// TIA Portal project "Hardware" (V14)

(* hardware
DEVICE "ET 200S-Station_1"  ET 200S station
   slot 0: "Baugruppenträger_0"  Rail
   slot 2: "PLC_1"  IM151-8 CPU  6ES7 151-8AB00-0AB0  V2.7
      slot 1: "PROFINET-Schnittstelle_1"  PN-IO
         slot 1: "Port_1"  Port
         slot 2: "Port_2"  Port
         slot 3: "Port_3"  Port
   slot 4: "PM-E 24VDC_1"  PM-E 24VDC  6ES7 138-4CA01-0AA0
   slot 5: "4AI x I 2WIRE ST_1"  4AI x I 2WIRE ST  6ES7 134-4GD00-0AB0
   slot 6: "2AO x U ST_1"  2AO x U ST  6ES7 135-4FB01-0AB0
   slot 7: "8DI x 24VDC_1"  8DI x 24VDC  6ES7 131-4BF00-0AA0
   slot 8: "8DI x 24VDC_2"  8DI x 24VDC  6ES7 131-4BF00-0AA0
   slot 9: "8DI x 24VDC_3"  8DI x 24VDC  6ES7 131-4BF00-0AA0
   slot 10: "8DI x 24VDC_4"  8DI x 24VDC  6ES7 131-4BF00-0AA0
   slot 11: "8DO x 24VDC / 0.5A_1"  8DO x 24VDC / 0.5A  6ES7 132-4BF00-0AA0
   slot 12: "8DO x 24VDC / 0.5A_2"  8DO x 24VDC / 0.5A  6ES7 132-4BF00-0AA0
   slot 13: "8DO x 24VDC / 0.5A_3"  8DO x 24VDC / 0.5A  6ES7 132-4BF00-0AA0
   slot 14: "8DO x 24VDC / 0.5A_4"  8DO x 24VDC / 0.5A  6ES7 132-4BF00-0AA0
DEVICE "HMI_1"  TP 177B 6'' PN/DP
   slot 0: "TP 177B 6'' PN/DP"  TP 177B 6'' PN/DP  6AV6 642-0BA01-1AX1  11.0.2.0
   slot 1: "HMI_RT_1"  TP 177B 6'' PN/DP  6AV6 642-0BA01-1AX1  11.0.2.0
   slot 5: "HMI_1.IE_CP_1"  PROFINET Interface  11.0.0.0
      slot 1: "PROFINET Schnittstelle_1"  PROFINET Interface
         slot 1: "Port_1"  Port
   slot 7: "HMI_1.MPI/DP_CP_1"  MPI/DP Interface  11.0.0.0
DEVICE "S7-1200-Station_1"  S7-1200 Station
   slot 0: "Baugruppenträger_0"  S7-1200 Rack  Rack  V1.0
   slot 1: "PLC_2"  CPU 1214FC DC/DC/DC  6ES7 214-1AF40-0XB0  V4.2
   slot 2: "F-DI 8/16x24VDC_1"  SM 1226 F-DI8/16 x 24VDC  6ES7 226-6BA32-0XB0  V2.0
   slot 3: "AI 1xRTD_1"  AI1 x RTD signal board  6ES7 231-5PA30-0XB0  V2.0
   slot 3: "F-DQ 4x24VDC_1"  SM 1226 F-DQ4 x 24VDC  6ES7 226-6DA32-0XB0  V2.0
   slot 4: "AI 4x13BIT/AQ 2x14BIT_1"  6ES7 234-4HE32-0XB0  V2.0
*)

// ===== PLC "PLC_1"  IM151-8 CPU =====

VAR_GLOBAL   // PLC tag table "Standard-Variablentabelle"
   "Blinken" AT %A7.0 : Bool;
   "Sekundentakt" AT %M100.5 : Bool;
   "A_rot" AT %A9.6 : Bool;
   "A_gelb" AT %A9.7 : Bool;
   "A_gruen" AT %A10.0 : Bool;
   "F_rot" AT %A10.6 : Bool;
   "F_gruen" AT %A10.7 : Bool;
   "Tag_1" AT %M0.0 : Bool;
   "Zweisekundentakt" AT %M100.7 : Bool;
   "Tag_2" AT %M3.0 : Bool;
   "Tag_3" AT %MD12 : DWord;
   "Tag_4" AT %MD16 : DWord;
   "Tag_5" AT %MW20 : Int;
   "Tag_6" AT %MW21 : Int;
   "Tag_7" AT %MW30 : Int;
   "Tag_8" AT %M22.7 : Bool;
   "Tag_9" AT %M2.0 : Bool;
   "Tag_10" AT %EW272 : Int;
END_VAR

DATA_BLOCK "Tagbetrieb_fb_DB"   // DB2
{ S7_Optimized_Access := 'FALSE' }
VERSION : 0.1
// stored: InstanceOfName Tagbetrieb_fb
"Tagbetrieb_fb"
BEGIN
END_DATA_BLOCK

DATA_BLOCK "DB3_Farben"   // DB3
{ S7_Optimized_Access := 'FALSE' }
VERSION : 0.1
   VAR
      rot : Int;
      gruen : Int;
      blau : Int;
   END_VAR
BEGIN
END_DATA_BLOCK

DATA_BLOCK "Farben"   // DB4
{ S7_Optimized_Access := 'FALSE' }
VERSION : 0.1
   VAR
      Farben : Array[0..2, 0..9] of Real;
      Rot : Real;
      Blau : Real;
      Gelb : Real;
      index : Int;
      schreiben : Bool;
   END_VAR
BEGIN
END_DATA_BLOCK

DATA_BLOCK "Zu_1200"   // DB100
{ S7_Optimized_Access := 'FALSE' }
VERSION : 0.1
   VAR
      Gewicht_rot : Real;
      Gewicht_Gruen : Real;
      Gewicht_Blau : Real;
   END_VAR
BEGIN
END_DATA_BLOCK

DATA_BLOCK "Von_1200"   // DB101
{ S7_Optimized_Access := 'FALSE' }
VERSION : 0.1
   VAR
      Temperatur : Int;
   END_VAR
BEGIN
END_DATA_BLOCK

DATA_BLOCK "Variable"   // DB200
{ S7_Optimized_Access := 'FALSE' }
VERSION : 0.1
   VAR
      Abstand : Real;
      Gewicht_real : Real;
      Volumen : Real;
      Tag : Bool;
      Zeit : Int;
      Tag_H : Int;
      Tag_M : Int;
      Start_tag : Int;
      Nacht_H : Int;
      Nacht_M : Int;
      Start_Nacht : Int;
   END_VAR
BEGIN
END_DATA_BLOCK

FUNCTION_BLOCK "Tagbetrieb_fb"   // FB1, FBD
{ S7_Optimized_Access := 'FALSE' }
VERSION : 0.1
   VAR_INPUT
      Sekundentakt : Bool;
   END_VAR
   VAR_OUTPUT
      Auto_rot : Bool;
      Auto_gelb : Bool;
      Auto_gruen : Bool;
      FG_rot : Bool;
      FG_gruen : Bool;
   END_VAR
   VAR
      S5 : Bool;
   END_VAR
   VAR_TEMP
      S1 : Bool;
      S2 : Bool;
      S3 : Bool;
      S4 : Bool;
      Zaehler : Int;
   END_VAR
BEGIN

REGION Network 1
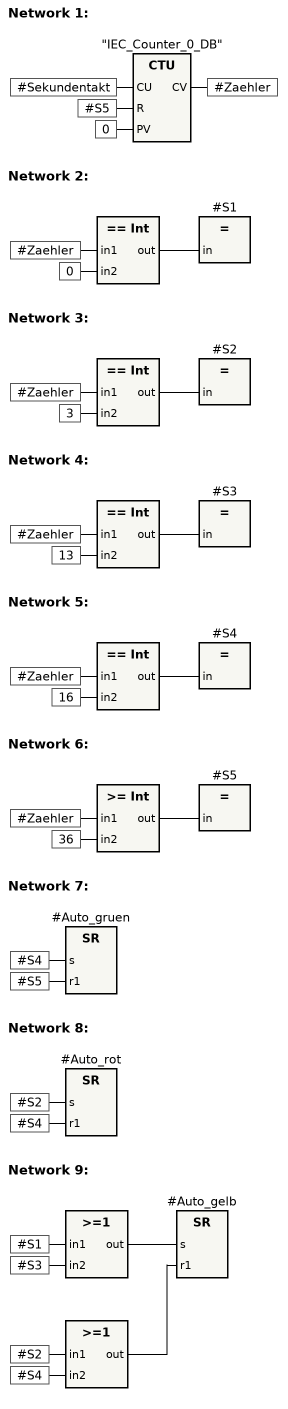
   "IEC_Counter_0_DB".CTU(CU := #Sekundentakt, R := #S5, PV := 0, CV => #Zaehler);
END_REGION

REGION Network 2
   #S1 := #Zaehler = 0;
END_REGION

REGION Network 3
   #S2 := #Zaehler = 3;
END_REGION

REGION Network 4
   #S3 := #Zaehler = 13;
END_REGION

REGION Network 5
   #S4 := #Zaehler = 16;
END_REGION

REGION Network 6
   #S5 := #Zaehler >= 36;
END_REGION

REGION Network 7
   IF #S4 THEN
       #Auto_gruen := TRUE;   // SR flip-flop
   END_IF;
   IF #S5 THEN #Auto_gruen := FALSE; END_IF;
END_REGION

REGION Network 8
   IF #S2 THEN
       #Auto_rot := TRUE;   // SR flip-flop
   END_IF;
   IF #S4 THEN #Auto_rot := FALSE; END_IF;
END_REGION

REGION Network 9
   IF #S1 OR #S3 THEN
       #Auto_gelb := TRUE;   // SR flip-flop
   END_IF;
   IF #S2 OR #S4 THEN #Auto_gelb := FALSE; END_IF;
END_REGION

REGION Network 10
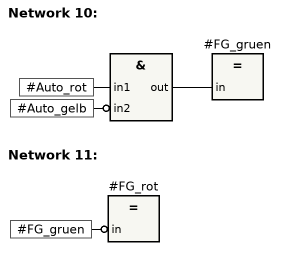
   #FG_gruen := #Auto_rot AND NOT #Auto_gelb;
END_REGION

REGION Network 11
   #FG_rot := NOT #FG_gruen;
END_REGION
END_FUNCTION_BLOCK

FUNCTION "Tagbetrieb" : Void   // FC1, FBD
{ S7_Optimized_Access := 'FALSE' }
VERSION : 0.1
   VAR_INPUT
      Sekundentakt : Bool;
   END_VAR
   VAR_OUTPUT
      Auto_rot : Bool;
      Auto_gelb : Bool;
      Auto_gruen : Bool;
      FG_rot : Bool;
      FG_gruen : Bool;
   END_VAR
   VAR_TEMP
      S1 : Bool;
      S2 : Bool;
      S3 : Bool;
      S4 : Bool;
      S5 : Bool;
      Zaehler : Int;
   END_VAR
BEGIN

REGION Network 1
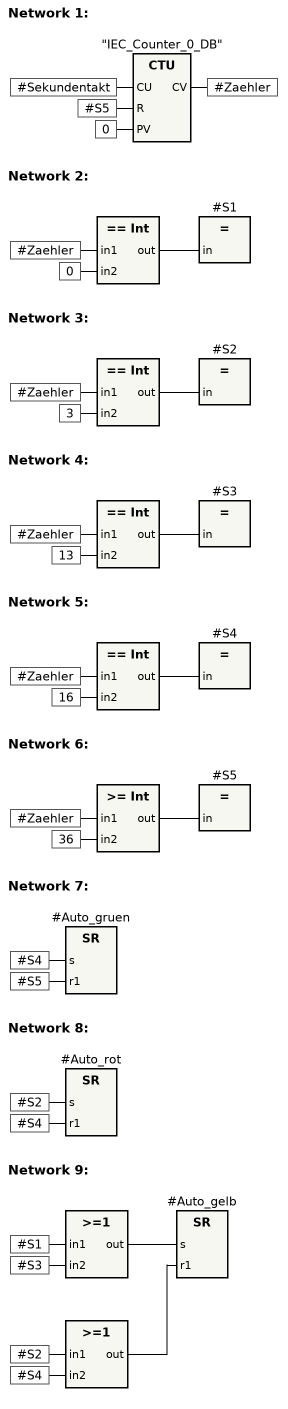
   "IEC_Counter_0_DB".CTU(CU := #Sekundentakt, R := #S5, PV := 0, CV => #Zaehler);
END_REGION

REGION Network 2
   #S1 := #Zaehler = 0;
END_REGION

REGION Network 3
   #S2 := #Zaehler = 3;
END_REGION

REGION Network 4
   #S3 := #Zaehler = 13;
END_REGION

REGION Network 5
   #S4 := #Zaehler = 16;
END_REGION

REGION Network 6
   #S5 := #Zaehler >= 36;
END_REGION

REGION Network 7
   IF #S4 THEN
       #Auto_gruen := TRUE;   // SR flip-flop
   END_IF;
   IF #S5 THEN #Auto_gruen := FALSE; END_IF;
END_REGION

REGION Network 8
   IF #S2 THEN
       #Auto_rot := TRUE;   // SR flip-flop
   END_IF;
   IF #S4 THEN #Auto_rot := FALSE; END_IF;
END_REGION

REGION Network 9
   IF #S1 OR #S3 THEN
       #Auto_gelb := TRUE;   // SR flip-flop
   END_IF;
   IF #S2 OR #S4 THEN #Auto_gelb := FALSE; END_IF;
END_REGION

REGION Network 10
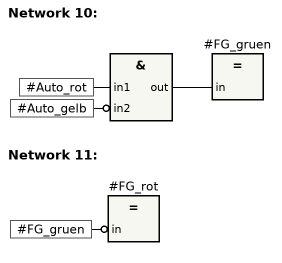
   #FG_gruen := #Auto_rot AND NOT #Auto_gelb;
END_REGION

REGION Network 11
   #FG_rot := NOT #FG_gruen;
END_REGION
END_FUNCTION

FUNCTION "Nachtbetrieb" : Void   // FC2, FBD
{ S7_Optimized_Access := 'FALSE' }
VERSION : 0.1
   VAR_INPUT
      Zweisekundentakt : Bool;
   END_VAR
   VAR_OUTPUT
      Auto_rot : Bool;
      Auto_gelb : Bool;
      Auto_gruen : Bool;
      FG_rot : Bool;
      FG_gruen : Bool;
   END_VAR
BEGIN

REGION Network 1
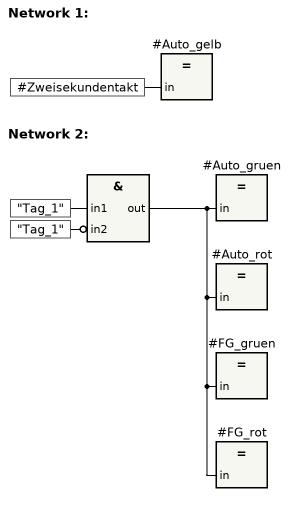
   #Auto_gelb := #Zweisekundentakt;
END_REGION

REGION Network 2
   #Auto_gruen := "Tag_1" AND NOT "Tag_1";
   #Auto_rot := #Auto_gruen;
   #FG_gruen := #Auto_gruen;
   #FG_rot := #Auto_gruen;
END_REGION
END_FUNCTION

FUNCTION "Minuten_des_Tages" : Int   // FC3, FBD
{ S7_Optimized_Access := 'FALSE' }
VERSION : 0.1
   VAR_INPUT
      Std : Byte;
      Min : Byte;
   END_VAR
   VAR_TEMP
      Std_w : Word;
      Std_i : Int;
      Min_w : Word;
      Min_i : Int;
      std_mal_60 : Int;
   END_VAR
BEGIN

REGION Network 1
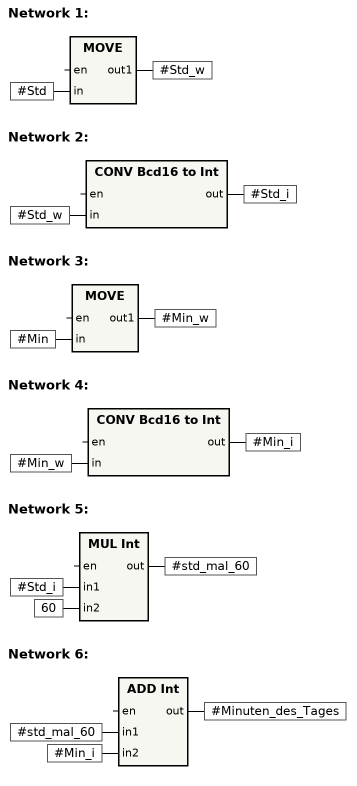
   #Std_w := #Std;
END_REGION

REGION Network 2
   #Std_i := BCD16_TO_INT(#Std_w);
END_REGION

REGION Network 3
   #Min_w := #Min;
END_REGION

REGION Network 4
   #Min_i := BCD16_TO_INT(#Min_w);
END_REGION

REGION Network 5
   #std_mal_60 := #Std_i * 60;
END_REGION

REGION Network 6
   #Minuten_des_Tages := #std_mal_60 + #Min_i;
END_REGION
END_FUNCTION

FUNCTION "Zeit_Rechnen" : Int   // FC4, FBD
{ S7_Optimized_Access := 'FALSE' }
VERSION : 0.1
   VAR_INPUT
      H : Int;
      "M" : Int;
   END_VAR
   VAR_TEMP
      H_mal_60 : Int;
   END_VAR
BEGIN

REGION Network 1
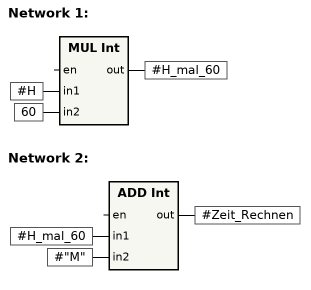
   #H_mal_60 := #H * 60;
END_REGION

REGION Network 2
   #Zeit_Rechnen := #H_mal_60 + #"M";
END_REGION
END_FUNCTION

FUNCTION "Vol_Zylinder" : Real   // FC5, SCL
{ S7_Optimized_Access := 'FALSE' }
VERSION : 0.1
   VAR_INPUT
      Durchmesser : Int;
      Hoehe : DInt;
   END_VAR
BEGIN
   IF #Durchmesser > 0 AND #Hoehe > 0 THEN
       #Vol_Zylinder := SQR(INT_TO_REAL(#Durchmesser)) * 0.785 * DINT_TO_REAL(#Hoehe);
   ELSE
       #Vol_Zylinder := -1.0;
   END_IF;
END_FUNCTION

FUNCTION "Induktive_sensor" : Real   // FC6, SCL
{ S7_Optimized_Access := 'FALSE' }
VERSION : 0.1
   VAR_INPUT
      value_sensor : Int;
   END_VAR
BEGIN
   IF #value_sensor <= -4800 THEN
       #Induktive_sensor := -1.0;

   ELSIF #value_sensor <> 0 AND #value_sensor > -4800 THEN
       #Induktive_sensor := (100 - INT_TO_REAL(#value_sensor)) / 490;
   ELSE
       #Induktive_sensor := -1.0;
   END_IF;
END_FUNCTION

FUNCTION "Gewicht_Zyl" : Real   // FC7, SCL
{ S7_Optimized_Access := 'FALSE' }
VERSION : 0.1
   VAR_INPUT
      Vol_Zylinder : Real;
      Dichte : Real;
   END_VAR
BEGIN
   IF #Vol_Zylinder <> 0 AND #Dichte <> 0 AND #Vol_Zylinder > 0 AND #Dichte > 0 THEN
       #Gewicht_Zyl := #Vol_Zylinder * #Dichte;
   ELSE
       #Gewicht_Zyl := 0;
   END_IF;
END_FUNCTION

FUNCTION "Farben_mischen" : Void   // FC8, SCL
{ S7_Optimized_Access := 'FALSE' }
VERSION : 0.1
   VAR_INPUT
      Schreiben : Bool;
      index : Int;
   END_VAR
   VAR_IN_OUT
      Farben : Array[0..2, 0..9] of Real;
      Rot : Real;
      Blau : Real;
      Gelb : Real;
   END_VAR
BEGIN
   IF #Schreiben THEN
       #Farben[0, #index] := #Rot;
       #Farben[1, #index] := #Blau;
       #Farben[2, #index] := #Gelb;
   ELSE
       #Rot  := #Farben[0, #index];
       #Blau := #Farben[1, #index];
       #Gelb := #Farben[2, #index];
   END_IF;
END_FUNCTION

FUNCTION "Masse_der_farben" : Real   // FC9, FBD
{ S7_Optimized_Access := 'FALSE' }
VERSION : 0.1
   VAR_INPUT
      Volumen : Int;
      Temperatur_mal_10 : Int;
   END_VAR
   VAR_TEMP
      Volumen_di : DInt;
      Volumen_r : Real;
      Temperatur_bezug : Int;
      Temperatur_bezug_di : DInt;
      Temperatur_bezug_r : Real;
      Gewichtzunahme : Real;
      Faktor : Real;
   END_VAR
BEGIN

REGION Network 1
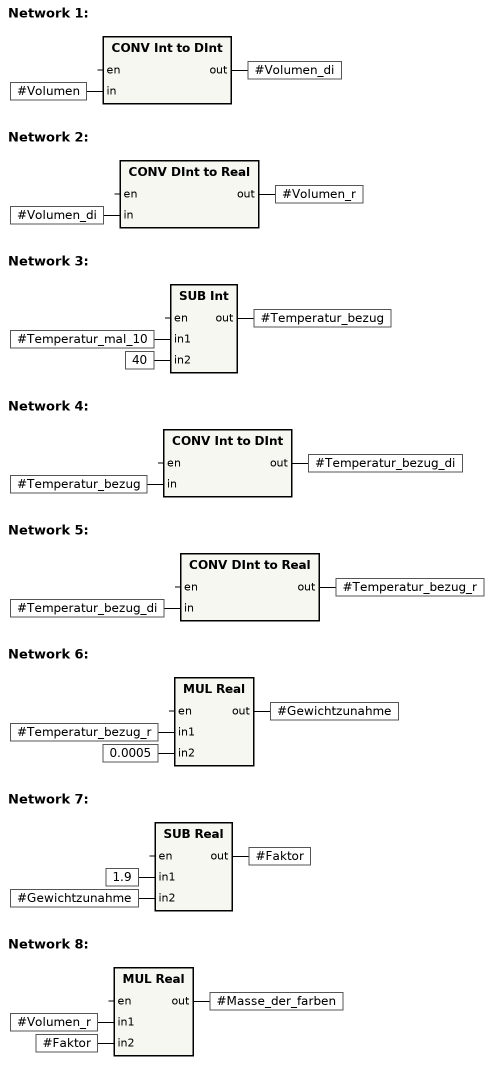
   #Volumen_di := INT_TO_DINT(#Volumen);
END_REGION

REGION Network 2
   #Volumen_r := DINT_TO_REAL(#Volumen_di);
END_REGION

REGION Network 3
   #Temperatur_bezug := #Temperatur_mal_10 - 40;
END_REGION

REGION Network 4
   #Temperatur_bezug_di := INT_TO_DINT(#Temperatur_bezug);
END_REGION

REGION Network 5
   #Temperatur_bezug_r := DINT_TO_REAL(#Temperatur_bezug_di);
END_REGION

REGION Network 6
   #Gewichtzunahme := #Temperatur_bezug_r * 0.0005;
END_REGION

REGION Network 7
   #Faktor := 1.9 - #Gewichtzunahme;
END_REGION

REGION Network 8
   #Masse_der_farben := #Volumen_r * #Faktor;
END_REGION
END_FUNCTION

ORGANIZATION_BLOCK "Main"   // OB1, FBD
TITLE = "Main Program Sweep (Cycle)"
{ S7_Optimized_Access := 'FALSE' }
VERSION : 0.1
   VAR_TEMP
      OB1_EV_CLASS : Byte;   // Bits 0-3 = 1 (Coming event), Bits 4-7 = 1 (Event class 1)
      OB1_SCAN_1 : Byte;   // 1 (Cold restart scan 1 of OB 1), 3 (Scan 2-n of OB 1)
      OB1_PRIORITY : Byte;   // Priority of OB Execution
      OB1_OB_NUMBR : Byte;   // 1 (Organization block 1, OB1)
      OB1_RESERVED_1 : Byte;   // Reserved for system
      OB1_RESERVED_2 : Byte;   // Reserved for system
      OB1_PREV_CYCLE : Int;   // Cycle time of previous OB1 scan (milliseconds)
      OB1_MIN_CYCLE : Int;   // Minimum cycle time of OB1 (milliseconds)
      OB1_MAX_CYCLE : Int;   // Maximum cycle time of OB1 (milliseconds)
      OB1_DATE_TIME : Date_And_Time;   // Date and time OB1 started
   END_VAR
BEGIN

REGION Network 1
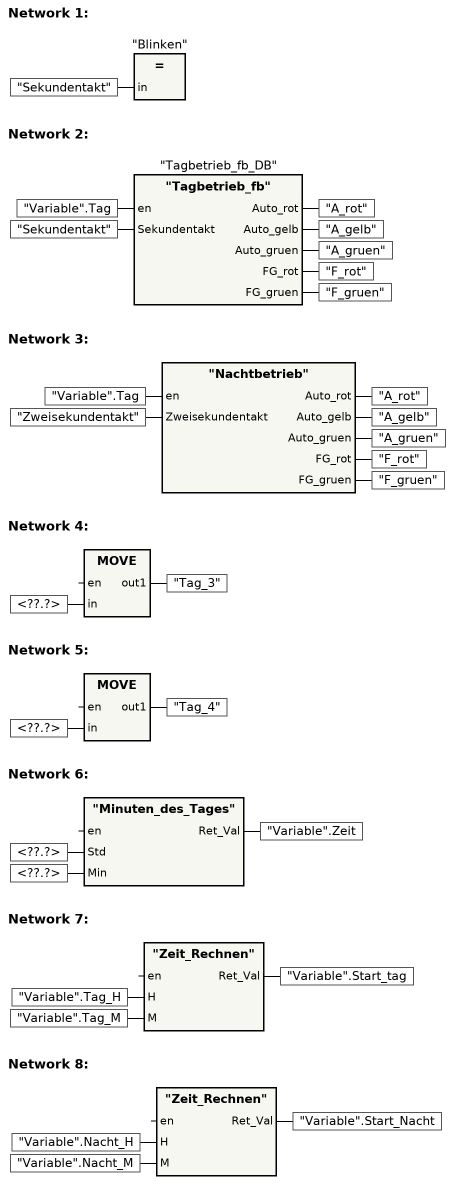
   "Blinken" := "Sekundentakt";
END_REGION

REGION Network 2
   IF "Variable".Tag THEN
       "Tagbetrieb_fb_DB"(Sekundentakt := "Sekundentakt",   // "Tagbetrieb_fb"
                          Auto_rot => "A_rot",
                          Auto_gelb => "A_gelb",
                          Auto_gruen => "A_gruen",
                          FG_rot => "F_rot",
                          FG_gruen => "F_gruen");
   END_IF;
END_REGION

REGION Network 3
   IF "Variable".Tag THEN
       "Nachtbetrieb"(Zweisekundentakt := "Zweisekundentakt",
                      Auto_rot => "A_rot",
                      Auto_gelb => "A_gelb",
                      Auto_gruen => "A_gruen",
                      FG_rot => "F_rot",
                      FG_gruen => "F_gruen");
   END_IF;
END_REGION

REGION Network 4
   "Tag_3" := <??.?>;
END_REGION

REGION Network 5
   "Tag_4" := <??.?>;
END_REGION

REGION Network 6
   "Variable".Zeit := "Minuten_des_Tages"(Std := <??.?>, Min := <??.?>);
END_REGION

REGION Network 7
   "Variable".Start_tag := "Zeit_Rechnen"(H := "Variable".Tag_H, "M" := "Variable".Tag_M);
END_REGION

REGION Network 8
   "Variable".Start_Nacht := "Zeit_Rechnen"(H := "Variable".Nacht_H, "M" := "Variable".Nacht_M);
END_REGION

REGION Network 9
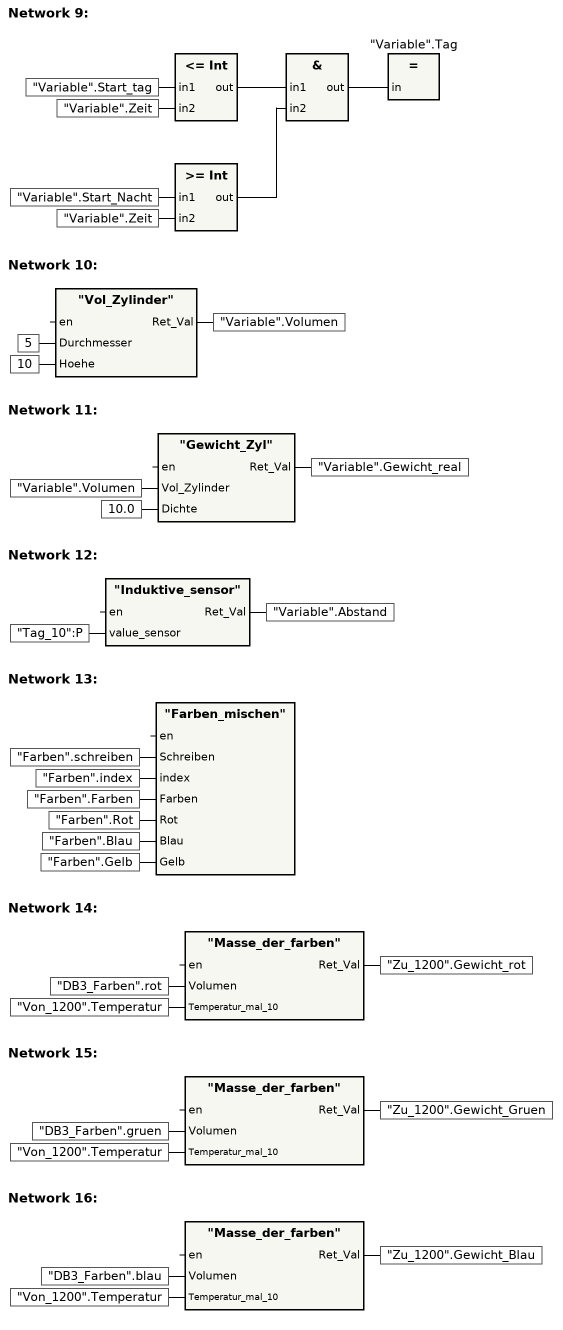
   "Variable".Tag := ("Variable".Start_tag <= "Variable".Zeit) AND ("Variable".Start_Nacht >= "Variable".Zeit);
END_REGION

REGION Network 10
   "Variable".Volumen := "Vol_Zylinder"(Durchmesser := 5, Hoehe := 10);
END_REGION

REGION Network 11
   "Variable".Gewicht_real := "Gewicht_Zyl"(Vol_Zylinder := "Variable".Volumen, Dichte := 10.0);
END_REGION

REGION Network 12
   "Variable".Abstand := "Induktive_sensor"(value_sensor := "Tag_10":P);
END_REGION

REGION Network 13
   "Farben_mischen"(Schreiben := "Farben".schreiben,
                    index := "Farben".index,
                    Farben := "Farben".Farben,
                    Rot := "Farben".Rot,
                    Blau := "Farben".Blau,
                    Gelb := "Farben".Gelb);
END_REGION

REGION Network 14
   "Zu_1200".Gewicht_rot := "Masse_der_farben"(Volumen := "DB3_Farben".rot,
                           Temperatur_mal_10 := "Von_1200".Temperatur);
END_REGION

REGION Network 15
   "Zu_1200".Gewicht_Gruen := "Masse_der_farben"(Volumen := "DB3_Farben".gruen,
                           Temperatur_mal_10 := "Von_1200".Temperatur);
END_REGION

REGION Network 16
   "Zu_1200".Gewicht_Blau := "Masse_der_farben"(Volumen := "DB3_Farben".blau,
                           Temperatur_mal_10 := "Von_1200".Temperatur);
END_REGION
END_ORGANIZATION_BLOCK

// ===== PLC "PLC_2"  CPU 1214FC DC/DC/DC =====

VAR_GLOBAL   // PLC tag table "Standard-Variablentabelle"
   "System_Byte" AT %MB1 : Byte;
   "FirstScan" AT %M1.0 : Bool;
   "DiagStatusUpdate" AT %M1.1 : Bool;
   "AlwaysTRUE" AT %M1.2 : Bool;
   "AlwaysFALSE" AT %M1.3 : Bool;
   "Clock_Byte" AT %MB100 : Byte;
   "Clock_10Hz" AT %M100.0 : Bool;
   "Clock_5Hz" AT %M100.1 : Bool;
   "Clock_2.5Hz" AT %M100.2 : Bool;
   "Clock_2Hz" AT %M100.3 : Bool;
   "Clock_1.25Hz" AT %M100.4 : Bool;
   "Clock_1Hz" AT %M100.5 : Bool;
   "Clock_0.625Hz" AT %M100.6 : Bool;
   "Clock_0.5Hz" AT %M100.7 : Bool;
   "System_Byte(1)" AT %MB0 : Byte;
   "Tag_1" AT %EW80 : Word;
   "Tag_2" AT %MW80 : Word;
   "Tag_3" AT %MD40 : Real;
   "Tag_4" AT %M3.0 : Bool;
   "Tag_5" AT %MD10 : DWord;
   "Tag_6" AT %MD11 : Real;
   "Tag_7" AT %MD12 : Real;
END_VAR

DATA_BLOCK "Main_Safety_RTG1_DB"   // DB1, F_DB
{ S7_Optimized_Access := 'TRUE' }
NAME : FUSI
VERSION : 0.1
// stored: InstanceOfName Main_Safety_RTG1
"Main_Safety_RTG1"
BEGIN
END_DATA_BLOCK

DATA_BLOCK "FB_datenaustausch_DB"   // DB6
{ S7_Optimized_Access := 'FALSE' }
VERSION : 0.1
// stored: InstanceOfName FB_datenaustausch
"FB_datenaustausch"
BEGIN
END_DATA_BLOCK

DATA_BLOCK "Von_300"   // DB100
{ S7_Optimized_Access := 'FALSE' }
VERSION : 0.1
   VAR
      Gewicht_rot : Real;
      Gewicht_Gruen : Real;
      Gewicht_blau : Real;
   END_VAR
BEGIN
END_DATA_BLOCK

DATA_BLOCK "Zu_300"   // DB101
{ S7_Optimized_Access := 'FALSE' }
VERSION : 0.1
   VAR
      Temperatur : Int;
   END_VAR
BEGIN
END_DATA_BLOCK

FUNCTION_BLOCK "Main_Safety_RTG1"   // FB1, F_FBD
{ S7_Optimized_Access := 'TRUE' }
VERSION : 0.1
BEGIN
END_FUNCTION_BLOCK

FUNCTION_BLOCK "FB_datenaustausch"   // FB99, FBD
{ S7_Optimized_Access := 'FALSE' }
VERSION : 0.1
   VAR_OUTPUT
      Fehler_uebetragen : Bool;
   END_VAR
   VAR
      Senden_aktiv : Bool;
      Senden_fertig : Bool;
      Empfangen_aktiv : Bool;
      Empfangen_fertig : Bool;
   END_VAR
   VAR_TEMP
      Status_Senden : Word;
      Status_empfangen : Word;
      Fehler_Senden : Bool;
      Fehler_Empfangen : Bool;
   END_VAR
BEGIN

REGION Network 1
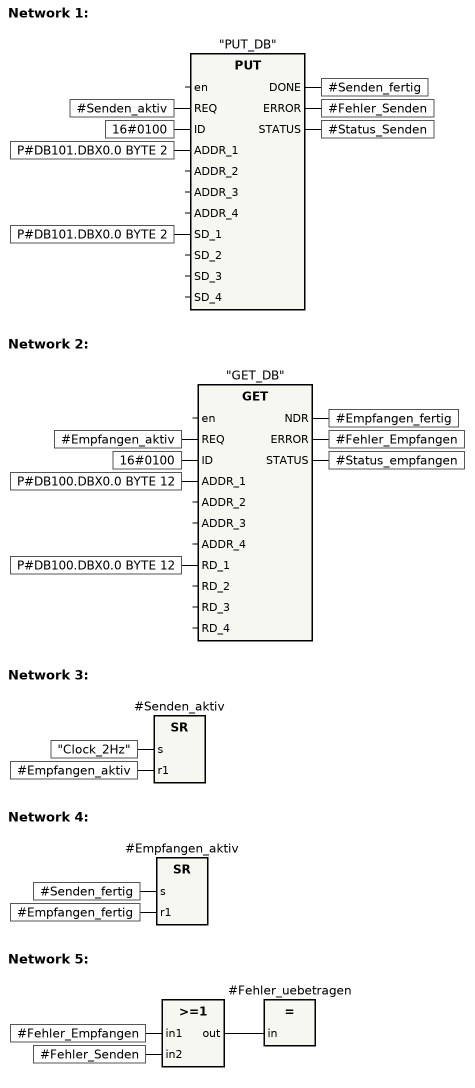
   "PUT_DB"(REQ := #Senden_aktiv,   // PUT
            ID := 16#0100,
            ADDR_1 := P#DB101.DBX0.0 BYTE 2,
            SD_1 := P#DB101.DBX0.0 BYTE 2,
            DONE => #Senden_fertig,
            ERROR => #Fehler_Senden,
            STATUS => #Status_Senden);
END_REGION

REGION Network 2
   "GET_DB"(REQ := #Empfangen_aktiv,   // GET
            ID := 16#0100,
            ADDR_1 := P#DB100.DBX0.0 BYTE 12,
            RD_1 := P#DB100.DBX0.0 BYTE 12,
            NDR => #Empfangen_fertig,
            ERROR => #Fehler_Empfangen,
            STATUS => #Status_empfangen);
END_REGION

REGION Network 3
   IF "Clock_2Hz" THEN
       #Senden_aktiv := TRUE;   // SR flip-flop
   END_IF;
   IF #Empfangen_aktiv THEN #Senden_aktiv := FALSE; END_IF;
END_REGION

REGION Network 4
   IF #Senden_fertig THEN
       #Empfangen_aktiv := TRUE;   // SR flip-flop
   END_IF;
   IF #Empfangen_fertig THEN #Empfangen_aktiv := FALSE; END_IF;
END_REGION

REGION Network 5
   #Fehler_uebetragen := #Fehler_Empfangen OR #Fehler_Senden;
END_REGION
END_FUNCTION_BLOCK

ORGANIZATION_BLOCK "Main"   // OB1, FBD, ProgramCycle
TITLE = "Main Program Sweep (Cycle)"
{ S7_Optimized_Access := 'TRUE' }
VERSION : 0.1
   VAR_INPUT
      Initial_Call : Bool;   // Initial call of this OB
      Remanence : Bool;   // =True, if remanent data are available
   END_VAR
BEGIN

REGION Network 1
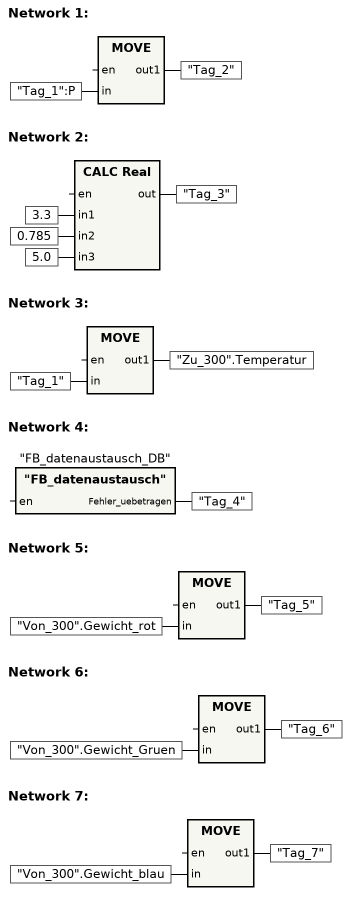
   "Tag_2" := "Tag_1":P;
END_REGION

REGION Network 2
   CALC(in1 := 3.3, in2 := 0.785, in3 := 5.0, out => "Tag_3");
END_REGION

REGION Network 3
   "Zu_300".Temperatur := "Tag_1";
END_REGION

REGION Network 4
   "FB_datenaustausch_DB"(Fehler_uebetragen => "Tag_4");   // "FB_datenaustausch"
END_REGION

REGION Network 5
   "Tag_5" := "Von_300".Gewicht_rot;
END_REGION

REGION Network 6
   "Tag_6" := "Von_300".Gewicht_Gruen;
END_REGION

REGION Network 7
   "Tag_7" := "Von_300".Gewicht_blau;
END_REGION
END_ORGANIZATION_BLOCK

(* ===== HMI "HMI_RT_1" =====
system functions are stored by id; their names below are inferred from use
connection "HMI_Verbindung_1": ETHERNET, SIMATIC S7 300/400 MPI
connection "HMI_Verbindung_2": ETHERNET, SIMATIC S7 1200

HMI tags "Standard-Variablentabelle"
   "Variable_Bildnummer" : UInt, internal
   "A_rot" : Bool = PLC A_rot AT %A9.6, 1 s
   "A_gelb" : Bool = PLC A_gelb AT %A9.7, 1 s
   "A_gruen" : Bool = PLC A_gruen AT %A10.0, 1 s
   "F_gruen" : Bool = PLC F_gruen AT %A10.7, 1 s
   "F_rot" : Bool = PLC F_rot AT %A10.6, 1 s
   "Variable_Tag_H" : Int = PLC Variable.Tag_H AT %DB200.DBW16, 1 s
   "Variable_Tag_M" : Int = PLC Variable.Tag_M AT %DB200.DBW18, 1 s
   "Variable_Nacht_H" : Int = PLC Variable.Nacht_H AT %DB200.DBW22, 1 s
   "Variable_Nacht_M" : Int = PLC Variable.Nacht_M AT %DB200.DBW24, 1 s
   "Variable_Abstand" : Real = PLC Variable.Abstand AT %DB200.DBD0, 1 s
   "Farben_Rot" : Real = PLC Farben.Rot AT %DB4.DBD120, 1 s
   "Farben_Blau" : Real = PLC Farben.Blau AT %DB4.DBD124, 1 s
   "Farben_Gelb" : Real = PLC Farben.Gelb AT %DB4.DBD128, 1 s
   "Farben_index" : Int = PLC Farben.index AT %DB4.DBW132, 1 s
   "Farben_schreiben" : Bool = PLC Farben.schreiben AT %DB4.DBX134.0, 1 s
   "DB3_Farben_rot" : Int = PLC DB3_Farben.rot AT %DB3.DBW0, 1 s
   "DB3_Farben_blau" : Int = PLC DB3_Farben.blau AT %DB3.DBW4, 1 s
   "Von_300_Gewicht_rot" : Real = PLC Von_300.Gewicht_rot AT %DB100.DBD0, 1 s
   "Von_300_Gewicht_Gruen" : Real = PLC Von_300.Gewicht_Gruen AT %DB100.DBD4, 1 s
   "Von_300_Gewicht_blau" : Real = PLC Von_300.Gewicht_blau AT %DB100.DBD8, 1 s
   "Zu_1200_Gewicht_Gruen" : Real = PLC Zu_1200.Gewicht_Gruen AT %DB100.DBD4, 1 s
   "Zu_1200_Gewicht_rot" : Real = PLC Zu_1200.Gewicht_rot AT %DB100.DBD0, 1 s
   "Zu_1200_Gewicht_Blau" : Real = PLC Zu_1200.Gewicht_Blau AT %DB100.DBD8, 1 s
   "DB3_Farben_gruen" : Int = PLC DB3_Farben.gruen AT %DB3.DBW2, 1 s

text list "Textliste_Bildnamen": 1 'Grundbild / base image'; 2 'Ampel / Trafic light'; 3 'Uhrzeit / Time'

text list "Farben": 0 'Orange'; 1 'Violett'; 2 'Hellblau'

screen "Grundbild" 320x200, template "Vorlage_1"
   on GenerateScreen: SetTag("Variable_Bildnummer", 1)
   TextField "HmiScreenItemData" at 21,55 size 179x36; Text 'Willkommen zum HMI_1 (TP 177B 6″ PN/DP)!'
   Button "Ampel" at 1,1 size 104x36; TextOff 'Ampel / Trafic light'
      on Release: ActivateScreen("Ampel", 0)
   Button "Uhrzeit" at 106,1 size 104x36; TextOff 'Uhrzeit / Time'
      on Release: ActivateScreen("Uhrzeit", 0)
   TextField "Textfeld_1" at 243,9 size 51x20; Text 'Sprache'
   Button "Schaltfläche_1" at 228,30 size 80x25; TextOff 'Deutsch'
      on Release: function_fb9197e8(L de-DE)
   Button "Schaltfläche_2" at 228,56 size 80x25; TextOff 'English'
      on Release: function_fb9197e8(L en-US)
   Button "Schaltfläche_3" at 0,124 size 160x25; TextOff 'Farben'
      on Click: ActivateScreen("Farben", 0)

Template "Vorlage_1" 320x200
   Button "Beenden" at 267,150 size 51x47; TextOff 'Beenden / Operate'; TextOn 'Beenden / Finish'; PictureOff "ExitRuntime_TP_177B_6_PNDP"; PictureOn "ExitRuntime_TP_177B_6_PNDP"
      on Release: StopRuntime(0)
   Button "Template_Button" at 214,150 size 51x47; TextOff 'Text'
   Button "Template_Button_1" at 160,150 size 51x47; TextOff 'Text'
   Button "Template_Button_2" at 107,150 size 51x47; TextOff 'Text'
   Button "Template_Button_3" at 54,150 size 51x47; TextOff 'Text'
   Button "Startbild" at 1,150 size 51x47; TextOff 'Startbild / Home'; PictureOff "NavigateHome_TP_177B_6_PNDP"; PictureOn "NavigateHome_TP_177B_6_PNDP"
      on Release: ActivateScreen("Grundbild", 0)

screen "Ampel" 320x200, template "Vorlage_1"
   on GenerateScreen: SetTag("Variable_Bildnummer", 2)
   GraphicView "Grafikanzeige_1" at 0,1 size 319x148; Picture "strasse"
   Group "Group" at 170,4 size 60x25
   Group "Group_1" at 83,119 size 60x25
   Group "Group_2" at 188,106 size 25x43
   Group "Group_3" at 110,1 size 25x43
   Circle "Kreis_1" at 173,7 size 18x18
      Visibility <- "A_rot"
   Circle "Kreis_2" at 192,7 size 18x18
      Appearance <- "A_gelb"
   Circle "Kreis_3" at 211,8 size 18x18
      Visibility <- "A_gruen"
   Circle "Kreis_4" at 122,122 size 18x18
      Visibility <- "A_rot"
   Circle "Kreis_5" at 103,122 size 18x18
      Appearance <- "A_gelb"
   Circle "Kreis_6" at 84,123 size 18x18
      Visibility <- "A_gruen"
   Circle "Kreis_9" at 192,107 size 18x18
      Visibility <- "F_gruen"
   Circle "Kreis_7" at 192,127 size 18x18
      Visibility <- "F_rot"
   Circle "Kreis_8" at 114,25 size 18x18
      Visibility <- "F_gruen"
   Circle "Kreis_10" at 114,5 size 18x18
      Visibility <- "F_rot"

screen "Uhrzeit" 320x200, template "Vorlage_1"
   on GenerateScreen: SetTag("Variable_Bildnummer", 3)
   Button "Zurück" at 1,1 size 104x36; TextOff 'Zurück / back'
      on Release: ActivateScreen("Grundbild", 0)
   TextField "Textfeld_1" at 18,42 size 31x20; Text 'Tag: / day'
   IOField "EA-Feld_1" at 60,42 size 17x20; FormatPattern 99
      ProcessValue <- "Variable_Tag_H"
   TextField "Textfeld_2" at 77,42 size 10x20; Text ':'
   IOField "EA-Feld_2" at 87,42 size 17x20; FormatPattern 99
      ProcessValue <- "Variable_Tag_M"
   TextField "Textfeld_3" at 105,42 size 42x20; Text 'Uhr / o'clock'
   TextField "Textfeld_4" at 19,72 size 41x20; Text 'Nacht: / night'
   IOField "EA-Feld_3" at 61,72 size 17x20; FormatPattern 99
      ProcessValue <- "Variable_Nacht_H"
   TextField "Textfeld_5" at 78,72 size 10x20; Text ':'
   IOField "EA-Feld_4" at 88,72 size 17x20; FormatPattern 99
      ProcessValue <- "Variable_Nacht_M"
   TextField "Textfeld_6" at 106,72 size 42x20; Text 'Uhr / o'clock'

screen "Abstandbild" 320x200
   Gauge "Zeigerinstrument_1" at 114,0 size 200x200; CaptionText 'Abstand'; UnitText 'mm'
      ProcessValue <- "Variable_Abstand"
   Button "Schaltfläche_1" at 5,167 size 80x25; TextOff 'Grundbild'

screen "Farben" 320x200
   Button "Schaltfläche_1" at 0,176 size 150x24; TextOff 'Grundbild'
      on Click: ActivateScreen("Grundbild", 0)
   TextField "Textfeld_1" at 19,20 size 29x20; Text 'Rot'
   TextField "Textfeld_2" at 19,44 size 29x20; Text 'Blau'
   TextField "Textfeld_3" at 19,73 size 29x20; Text 'Gelb'
   TextField "Textfeld_4" at 19,99 size 35x20; Text 'Index'
   IOField "EA-Feld_1" at 54,20 size 80x20; FormatPattern s999999999.999
      ProcessValue <- "Farben_Rot"
   IOField "EA-Feld_2" at 54,48 size 80x20; FormatPattern s999999999.999
      ProcessValue <- "Farben_Blau"
   IOField "EA-Feld_3" at 54,75 size 80x20; FormatPattern s999999999.999
      ProcessValue <- "Farben_Gelb"
   IOField "EA-Feld_4" at 54,100 size 80x20; FormatPattern s99999
      ProcessValue <- "Farben_index"
   Button "Schaltfläche_2" at 56,134 size 80x25; TextOff 'Schreiben'
      on Click: InvertBit("Farben_schreiben")
      Appearance <- "Farben_schreiben"
   SymbolicIOField "Symbolisches EA-Feld_1" at 145,100 size 119x22; TextOff '0'; TextOn '1'; TextList "Farben"
      ProcessValue <- "Farben_index"

screen "Kontrollbild" 320x200
   TextField "Textfeld_1" at 13,28 size 30x20; Text 'grun'
   TextField "Textfeld_2" at 144,28 size 82x20; Text 'ausgabe grun'
   TextField "Textfeld_3" at 14,53 size 29x20; Text 'rot'
   TextField "Textfeld_4" at 13,79 size 29x20; Text 'Blau'
   TextField "Textfeld_5" at 147,80 size 81x20; Text 'Ausgabe Blau'
   TextField "Textfeld_6" at 146,52 size 75x20; Text 'ausgabe Rot'
   IOField "EA-Feld_2" at 228,52 size 80x20; FormatPattern s999999999.999
      ProcessValue <- "Von_300_Gewicht_rot"
   IOField "EA-Feld_3" at 229,27 size 80x20; FormatPattern s999999999.999
      ProcessValue <- "Von_300_Gewicht_Gruen"
   IOField "EA-Feld_4" at 229,81 size 80x20; FormatPattern s999999999.999
      ProcessValue <- "Von_300_Gewicht_blau"
   IOField "EA-Feld_1" at 47,30 size 93x20; FormatPattern s99999
      ProcessValue <- "DB3_Farben_gruen"
   IOField "EA-Feld_5" at 46,53 size 94x20; FormatPattern s99999
      ProcessValue <- "DB3_Farben_rot"
   IOField "EA-Feld_6" at 46,80 size 95x20; FormatPattern s99999
      ProcessValue <- "DB3_Farben_blau"
*)